//==================================================================================================
//								RJM Maszyny sp. z o.o.
//									14.06.2022
//	FB posredniczący pomiędzy FB a logerem alarmów  
// 	v1.0	|| TC v 3.1.4024.22		|| - pierwsza wersja
//==================================================================================================
FUNCTION_BLOCK FB_Silownik_Kontrola_Komunikacja EXTENDS FB_LogowanieBledow_ElementWykonawczy
VAR_INPUT
END_VAR
VAR_OUTPUT
END_VAR
VAR
	
END_VAR

METHOD DefinicjaTabeliZdarzen_1031_Niemiecki : BOOL
VAR_INPUT
	arrTablicaDefinicjiZdarzenOpis			: REFERENCE TO ARRAY [1..GVL_LogowanieBledow_Stale.MAX_ILOSC_ZDARZEN] OF DUT_LogowanieBledow_ZdarzenieOpis;

END_VAR
arrTablicaDefinicjiZdarzenOpis [iStartId+0].sOpis	:= 'DE - zbyt dlugi czas w stronę końca';
arrTablicaDefinicjiZdarzenOpis [iStartId+1].sOpis	:= 'DE - zbyt dlugi czas w stronę początku';
arrTablicaDefinicjiZdarzenOpis [iStartId+2].sOpis	:= 'DE - utrata pozycji 0';
arrTablicaDefinicjiZdarzenOpis [iStartId+3].sOpis	:= 'DE - utrata pozycji MAX';
arrTablicaDefinicjiZdarzenOpis [iStartId+4].sOpis	:= 'DE - blad ustawienia czujnikow - dwa czujniki aktywne';
arrTablicaDefinicjiZdarzenOpis [iStartId+5].sOpis	:= 'DE - blad ustawiania ustawienia czujników - zamienione miejscami';
END_METHOD

METHOD DefinicjaTabeliZdarzen_1033_Angielski : BOOL
VAR_INPUT
	arrTablicaDefinicjiZdarzenOpis			: REFERENCE TO ARRAY [1..GVL_LogowanieBledow_Stale.MAX_ILOSC_ZDARZEN] OF DUT_LogowanieBledow_ZdarzenieOpis;

END_VAR
arrTablicaDefinicjiZdarzenOpis [iStartId+0].sOpis	:= 'EN - zbyt dlugi czas w stronę końca';
arrTablicaDefinicjiZdarzenOpis [iStartId+1].sOpis	:= 'EN - zbyt dlugi czas w stronę początku';
arrTablicaDefinicjiZdarzenOpis [iStartId+2].sOpis	:= 'EN - utrata pozycji 0';
arrTablicaDefinicjiZdarzenOpis [iStartId+3].sOpis	:= 'EN - utrata pozycji MAX';
arrTablicaDefinicjiZdarzenOpis [iStartId+4].sOpis	:= 'EN - blad ustawienia czujnikow - dwa czujniki aktywne';
arrTablicaDefinicjiZdarzenOpis [iStartId+5].sOpis	:= 'EN - blad ustawiania ustawienia czujników - zamienione miejscami';
END_METHOD

METHOD DefinicjaTabeliZdarzen_1045_Polski : BOOL
VAR_INPUT
	arrTablicaDefinicjiZdarzenOpis			: REFERENCE TO ARRAY [1..GVL_LogowanieBledow_Stale.MAX_ILOSC_ZDARZEN] OF DUT_LogowanieBledow_ZdarzenieOpis;

END_VAR
arrTablicaDefinicjiZdarzenOpis [iStartId+0].sOpis	:= 'PL - zbyt dlugi czas w stronę końca';
arrTablicaDefinicjiZdarzenOpis [iStartId+1].sOpis	:= 'PL - zbyt dlugi czas w stronę początku';
arrTablicaDefinicjiZdarzenOpis [iStartId+2].sOpis	:= 'PL - utrata pozycji 0';
arrTablicaDefinicjiZdarzenOpis [iStartId+3].sOpis	:= 'PL - utrata pozycji MAX';
arrTablicaDefinicjiZdarzenOpis [iStartId+4].sOpis	:= 'PL - blad ustawienia czujnikow - dwa czujniki aktywne';
arrTablicaDefinicjiZdarzenOpis [iStartId+5].sOpis	:= 'PL - blad ustawiania ustawienia czujników - zamienione miejscami';
END_METHOD

METHOD DefinicjaTabeliZdarzen_Ogolna : BOOL
VAR_INPUT
	arrTablicaDefinicjiZdarzen				: REFERENCE TO ARRAY [1..GVL_LogowanieBledow_Stale.MAX_ILOSC_ZDARZEN] OF DUT_LogowanieBledow_Zdarzenie;
	arrTablicaDefinicjiZdarzenOpis			: REFERENCE TO ARRAY [1..GVL_LogowanieBledow_Stale.MAX_ILOSC_ZDARZEN] OF DUT_LogowanieBledow_ZdarzenieOpis;
	arrTablicaDefinicjiZdarzenStan			: REFERENCE TO ARRAY [1..GVL_LogowanieBledow_Stale.MAX_ILOSC_ZDARZEN] OF DUT_LogowanieBledow_ZdarzenieStan;

	iIdZdarzenia							: REFERENCE TO INT;
	iNrPodzespolu							: INT := 0;
	iNrPodelementu							: INT := 0;
	iNrElementu								: INT := 0;
END_VAR
//zbyt dlugi czas w stronę końca
	iIdZdarzenia										:= iIdZdarzenia + 1;
	arrTablicaDefinicjiZdarzen [iIdZdarzenia].iIdZdarzenia			:= iIdZdarzenia;
	arrTablicaDefinicjiZdarzen [iIdZdarzenia].byRodzajZdarzenia	:= 2;
	arrTablicaDefinicjiZdarzen [iIdZdarzenia].sKodBledu			:= '0001';
	arrTablicaDefinicjiZdarzen [iIdZdarzenia].sNrKomponentu		:= GenerujNrKomponentu (iNrPodzespolu := iNrPodzespolu, iNrPodelementu := iNrPodelementu, iNrElementu := iNrElementu); 
	arrTablicaDefinicjiZdarzenOpis [iIdZdarzenia].iIdZdarzenia 	:= iIdZdarzenia;
	arrTablicaDefinicjiZdarzenStan [iIdZdarzenia].iIdZdarzenia 	:= iIdZdarzenia;
	arrTablicaDefinicjiZdarzenStan [iIdZdarzenia].bAktywne			:= FALSE;
//zbyt dlugi czas w stronę początku	
	iIdZdarzenia										:= iIdZdarzenia + 1;
	arrTablicaDefinicjiZdarzen [iIdZdarzenia].iIdZdarzenia			:= iIdZdarzenia;
	arrTablicaDefinicjiZdarzen [iIdZdarzenia].byRodzajZdarzenia	:= 2;
	arrTablicaDefinicjiZdarzen [iIdZdarzenia].sKodBledu			:= '0002';
	arrTablicaDefinicjiZdarzen [iIdZdarzenia].sNrKomponentu		:= GenerujNrKomponentu (iNrPodzespolu := iNrPodzespolu, iNrPodelementu := iNrPodelementu, iNrElementu := iNrElementu); 
	arrTablicaDefinicjiZdarzenOpis [iIdZdarzenia].iIdZdarzenia 	:= iIdZdarzenia;
	arrTablicaDefinicjiZdarzenStan [iIdZdarzenia].iIdZdarzenia 	:= iIdZdarzenia;
	arrTablicaDefinicjiZdarzenStan [iIdZdarzenia].bAktywne			:= FALSE;
//utrata pozycji 0
	iIdZdarzenia										:= iIdZdarzenia + 1;
	arrTablicaDefinicjiZdarzen [iIdZdarzenia].iIdZdarzenia			:= iIdZdarzenia;
	arrTablicaDefinicjiZdarzen [iIdZdarzenia].byRodzajZdarzenia	:= 2;
	arrTablicaDefinicjiZdarzen [iIdZdarzenia].sKodBledu			:= '0003';
	arrTablicaDefinicjiZdarzen [iIdZdarzenia].sNrKomponentu 		:= GenerujNrKomponentu (iNrPodzespolu := iNrPodzespolu, iNrPodelementu := iNrPodelementu, iNrElementu := iNrElementu); 
	arrTablicaDefinicjiZdarzenOpis [iIdZdarzenia].iIdZdarzenia 	:= iIdZdarzenia;
	arrTablicaDefinicjiZdarzenStan [iIdZdarzenia].iIdZdarzenia 	:= iIdZdarzenia;
	arrTablicaDefinicjiZdarzenStan [iIdZdarzenia].bAktywne			:= FALSE;
//utrata pozycji MAX
	iIdZdarzenia										:= iIdZdarzenia + 1;
	arrTablicaDefinicjiZdarzen [iIdZdarzenia].iIdZdarzenia			:= iIdZdarzenia;
	arrTablicaDefinicjiZdarzen [iIdZdarzenia].byRodzajZdarzenia	:= 2;
	arrTablicaDefinicjiZdarzen [iIdZdarzenia].sKodBledu			:= '0004';
	arrTablicaDefinicjiZdarzen [iIdZdarzenia].sNrKomponentu 		:= GenerujNrKomponentu (iNrPodzespolu := iNrPodzespolu, iNrPodelementu := iNrPodelementu, iNrElementu := iNrElementu); 
	arrTablicaDefinicjiZdarzenOpis [iIdZdarzenia].iIdZdarzenia 	:= iIdZdarzenia;
	arrTablicaDefinicjiZdarzenStan [iIdZdarzenia].iIdZdarzenia 	:= iIdZdarzenia;
	arrTablicaDefinicjiZdarzenStan [iIdZdarzenia].bAktywne			:= FALSE;
//blad ustawienia czujnikow - dwa czujniki aktywne
	iIdZdarzenia										:= iIdZdarzenia + 1;
	arrTablicaDefinicjiZdarzen [iIdZdarzenia].iIdZdarzenia			:= iIdZdarzenia;
	arrTablicaDefinicjiZdarzen [iIdZdarzenia].byRodzajZdarzenia	:= 1;
	arrTablicaDefinicjiZdarzen [iIdZdarzenia].sKodBledu			:= '0005';
	arrTablicaDefinicjiZdarzen [iIdZdarzenia].sNrKomponentu 		:= GenerujNrKomponentu (iNrPodzespolu := iNrPodzespolu, iNrPodelementu := iNrPodelementu, iNrElementu := iNrElementu); 
	arrTablicaDefinicjiZdarzenOpis [iIdZdarzenia].iIdZdarzenia 	:= iIdZdarzenia;
	arrTablicaDefinicjiZdarzenStan [iIdZdarzenia].iIdZdarzenia 	:= iIdZdarzenia;
	arrTablicaDefinicjiZdarzenStan [iIdZdarzenia].bAktywne			:= FALSE;
//blad ustawiania ustawienia czujników - zamienione miejscami	
	iIdZdarzenia										:= iIdZdarzenia + 1;
	arrTablicaDefinicjiZdarzen [iIdZdarzenia].iIdZdarzenia			:= iIdZdarzenia;
	arrTablicaDefinicjiZdarzen [iIdZdarzenia].byRodzajZdarzenia	:= 1;
	arrTablicaDefinicjiZdarzen [iIdZdarzenia].sKodBledu			:= '0006';
	arrTablicaDefinicjiZdarzen [iIdZdarzenia].sNrKomponentu 		:= GenerujNrKomponentu (iNrPodzespolu := iNrPodzespolu, iNrPodelementu := iNrPodelementu, iNrElementu := iNrElementu); 
	arrTablicaDefinicjiZdarzenOpis [iIdZdarzenia].iIdZdarzenia 	:= iIdZdarzenia;
	arrTablicaDefinicjiZdarzenStan [iIdZdarzenia].iIdZdarzenia 	:= iIdZdarzenia;
	arrTablicaDefinicjiZdarzenStan [iIdZdarzenia].bAktywne			:= FALSE;
END_METHOD

END_FUNCTION_BLOCK

(* stored: Version 1.1.0.1, ProductVersion 3.1.4024.11
   POU FB_Silownik_Kontrola_Komunikacja: Id {6e1765c6-13ef-4cc8-af85-b94298696ee7}, SpecialFunc None
   Method DefinicjaTabeliZdarzen_1031_Niemiecki: Id {86e170c4-ab8f-448f-ade2-be1b5c03aa46}
   Method DefinicjaTabeliZdarzen_1033_Angielski: Id {312f69bd-29fe-40fb-abd4-3ca95737ef6e}
   Method DefinicjaTabeliZdarzen_1045_Polski: Id {1da6467f-9535-4281-b512-f948c9de2cca}
   Method DefinicjaTabeliZdarzen_Ogolna: Id {56182eaa-3642-491d-aa11-de8bc029eba9} *)
